Fanuc KAREL source: kt00130.KL

-- PROVISIONAL review KL for V770-1; original PC SHA256 f2284ad9a746849e67c246123334427e30416aec3c047ed213e22738f7f3bc2c
-- Incomplete behavior may be omitted. Consult companion uncertainty JSON. Do not deploy.
PROGRAM KT00130
%NOLOCKGROUP
VAR
  I1 : INTEGER
  I2 : INTEGER
  OUT : REAL
BEGIN
  -- UNRESOLVED_PC offsets 5-16; opcodes 2E,23
  -- UNRESOLVED_PC offsets 21-32; opcodes 2E,23
  -- UNRESOLVED_PC offsets 37-48; opcodes 2E,23
  -- UNRESOLVED_PC offsets 53-64; opcodes 2E,23
  -- UNRESOLVED_PC offsets 69-89; opcodes 21,21,55,64,23
  -- UNRESOLVED_PC offsets 94-98; opcodes 7F
END KT00130
